// TIA Portal V17 export
// export: Created 2025-03-10T13:09:25.930153Z, ExportSetting WithDefaults, DisplayName Totally Integrated Automation Portal, DisplayVersion V17 Update 8, DisplayName TIA Portal Openness, DisplayVersion V17 Update 8, DisplayName TIA Portal Version Control Interface, DisplayVersion V17, DisplayName SINAMICS Startdrive Advanced, DisplayVersion V17 SP2, DisplayName SINAMICS Startdrive G110M, G120, G120C, G120D, G120P, G115D, DisplayVersion V17 SP2, DisplayName SINAMICS Startdrive G130, G150, S120, S150, SINAMICS MV, S210, DisplayVersion V17 SP2, DisplayName STEP 7 Professional, DisplayVersion V17 Update 8, DisplayName SINUMERIK ONE STEP 7 Toolbox, DisplayVersion V17 Update 12, DisplayName SINUMERIK 840D sl STEP 7 Toolbox, DisplayVersion V17 Update 12, DisplayName STEP 7 Safety, DisplayVersion V17 Update 6, DisplayName WinCC Advanced, DisplayVersion V17 Update 8
DATA_BLOCK "LBP_TMLoadMT"   // DB1071
TITLE = Tool management / Gestión de herramientas / Werkzeugverwaltung
{ S7_Optimized_Access := 'FALSE'; DB_Accessible_From_OPC_UA := 'FALSE' }
AUTHOR : SINUMERIK
FAMILY : SINUMERIK_ONE
VERSION : 6.15
// Interface between user program and tool management, contains signals from/to Load/Unload magazine (multitool). / Interfaz entre programa de usuario y gestión de herramientas, contiene señales desde/hacia carga/descarga del almacén (Multitool). / Schnittstelle zwischen Anwenderprogramm und Werkzeugverwaltung, enthält Signale von/zu Laden/Entladen des Magazins (Multitool).
// stored: AutoNumber false, DBAccessibleFromOPCUA false, DBAccessibleFromWebserver true, InstanceOfName LBP_typeTMLoadMT, InstanceOfType UDT, IsOnlyStoredInLoadMemory false, IsWriteProtectedInAS false
"LBP_typeTMLoadMT"
   // VAR RETAIN
   //    MTIF : Array[1..16] of Struct
   //       DistanceCoding : Int;
   //       Places : Int;
   //       Distance : Real;
   //       MTNo : Int;
   //       PlaceNo : Int;
   //       Toolholder : Int;
   //       reserved : Array[1..3] of Int;
   //    END_STRUCT;
   // END_VAR
BEGIN
END_DATA_BLOCK
